{attribute addProperty BoxType "EP9224-0037-0017"}
{attribute addProperty Id "DPO_Inputs_ChannelAT %I*ARRAY[0..9] OF DPO_Inputs_Channel_AD3CD21C192240DPO_Inputs_DeviceAT %I*DPO_Inputs_Device_C2311DBA96120DPO_Outputs_ChannelAT %Q*ARRAY[0..12] OF DPO_Outputs_Channel_5760563F128160DPO_Outputs_DeviceAT %Q*DPO_Outputs_Device_6EB864581620WcStateAT %I*WcState_98A4DF7520.250InfoDataAT %I*InfoData_0BDED7BF144180"}
{attribute addProperty CRC "2418294593"}
{attribute addProperty SizeInBites "578"}
{attribute addProperty SizeInBytes "72.25"}
TYPE EP9224_2CE99204 :
STRUCT
	{attribute addProperty Name "DPO_Inputs_Channel"}
	DPO_Inputs_Channel : ARRAY[0..9] OF DPO_Inputs_Channel_AD3CD21C;
	{attribute addProperty Name "DPO_Inputs_Device"}
	DPO_Inputs_Device : DPO_Inputs_Device_C2311DBA;
	{attribute addProperty Name "DPO_Outputs_Channel"}
	DPO_Outputs_Channel : ARRAY[0..12] OF DPO_Outputs_Channel_5760563F;
	{attribute addProperty Name "DPO_Outputs_Device"}
	DPO_Outputs_Device : DPO_Outputs_Device_6EB86458;
	{attribute addProperty Name "WcState"}
	WcState : WcState_98A4DF75;
	{attribute addProperty Name "InfoData"}
	InfoData : InfoData_0BDED7BF;
END_STRUCT
END_TYPE

(* stored: Version 1.2.0.0, ProductVersion 3.1.4024.9
   DUT EP9224_2CE99204: Id {07174ed2-89d0-4373-80c7-ce0309b1d6e2} *)
